PROGRAM Welding_Robot
VAR
END_VAR

// =======================逻辑控制==========================
Robot_Simulink.stInput.t := t;											// 采样时间t与Simulink模型中的采样时间链接
//Hexapod_Robot.Model_Position := Robot_Simulink.stOutput.Disp_P;			// Simulink中的电机输出位移输入到控制模型
//Welding_Arm.Model_Position := Robot_Simulink.stOutput.Disp_P;			// Simulink中的电机输出位移输入到控制模型

END_PROGRAM

(* stored: Version 1.1.0.1, ProductVersion 3.1.4020.12
   POU Welding_Robot: Id {b66e518f-e7f0-493b-b5d2-0962412c8e91}, SpecialFunc None *)
